(* Logix 5000 project; controller cal1615 1756-L62 rev 16.20; software revision 16.05; part 26 of 78 *)
(* tags used below, declared in another part *)
   AFI : BOOL;   // Always False Bit
   FAULT : BOOL;   // Fault AFI
   p01_param_fan_zero_speed : REAL;
   p01_param_open_oven_exh_sp : REAL;
   p01_recipe_active : recipe;   // Active Recipe
   p01r02 : routine;   // System Misc Control
   p01r09_open_oven : BOOL;
   p01r09_pb_global_reset : BOOL;   // System Modes PB: Global Fault Reset
   p02_dint_from_hmi : hmi_dint;
   p11r02_shutdown_temp : BOOL;   // Zone 1 Misc Control Safe Shutdown Temperature
   p11r30 : routine;   // Zone 1 Temperature Control
   p11r30_request_heat : BOOL;   // Zone 1 Temperature Control Request Heat
   p12_ai_exhaust_rpm : REAL;   // Zone 2 Analog Input Exhaust Fan RPM
   p12_ai_lfl : REAL;   // Zone 2 Analog Input Lower Flash Limit
   p12_ao_exhaust_selected_speed : REAL;   // Zone 2 Analog Output Exhaust Fan VFD Selected Speed
   p12_di_burner_auto : BOOL;   // Zone 2 Digital Input Burner Auto
   p12_di_exh : acs800_di_normal;   // Zone 2 Digital Inputs Exhaust Fan
   p12_di_exh_fan_mtr_ts : BOOL;   // Zone 2 Digital Input Exhaust Fan Motor Thermostat OK
   p12_di_exh_flow_ok : BOOL;   // Zone 2 Digital Input Exhaust Flow OK
   p12_di_flame_on : BOOL;   // Zone 2 Digital Input Burner is On
   p12_di_fresh_air_clean : BOOL;   // Zone 2 Digital Input Fresh Air Filter Dirty
   p12_di_sp0 : BOOL;
   p12_di_tc01_bo : BOOL;   // Zone 2 Digital Input Control Thermocouple 1 Failure
   p12_di_tc02_bo : BOOL;   // Zone 2 Digital Input Control Thermocouple 2 Failure
   p12_di_zone_air_clean : BOOL;   // Zone 2 Digital Input Zone 2 Filter Dirty
   p12_do_exh : acs800_do_normal;   // Zone 2 Digital Output Exhaust Fan
   p12_param_lfl_hl : REAL;   // Zone 2 Parameter High LFL Limit
   p12_param_tc01_dev : REAL;   // Zone 2 Parameter Oven Temperature Deviation from Setpoint
   p12r01 : routine;   // Zone 2 Main
   p12r02_shutdown_temp : BOOL;   // Zone 2 Misc Control Safe Shutdown Temperature
   p12r20_safeties_ok : BOOL;   // Zone 2 Temperature Control Burner Safeties OK this Lightoff
   p12r20_state : DINT;   // Zone 2 Temperature Control State
   p12r30 : routine;   // Zone 2 Temperature Control
   p12r30_pb_zone_on : BOOL;   // Zone 2 Temperature Control PB: Start Zone Heat Control
   p12r30_pid_temp_sp_error : REAL;   // Zone 2 Temperature Control Setpoint/Process Variable Error (ABS)
   p12r30_request_deviation_warning : BOOL;   // Zone 2 Temperature Control Request Setpoint Deviation Warning
   p12r30_request_heat : BOOL;   // Zone 2 Temperature Control Request Heat
   p12r30_request_heat_last : BOOL;   // Zone 2 Temperature Control Request Heat Last Scan
   p12r30_request_manual : BOOL;   // Zone 2 Temperature Control Request Manual Control
   p12r30_timer_fault : TIMER[16];   // Zone 2 Temperature Control Fault Delay
   p12r30_timer_warning : TIMER[12];   // Zone 2 Temperature Control Warning Delay
   p12r31 : routine;   // Zone 2 Exhaust VFD
   p12r31_pb_start : BOOL;   // Zone 2 Exhaust VFD PB: Start
   p12r31_pb_stop : BOOL;   // Zone 2 Exhaust VFD PB: Stop
   p12r31_request_auto_run : BOOL;   // Zone 2 Exhaust Fan Run Request
   p12r31_run_permissive : BOOL;   // Zone 2 Exhaust VFD Run Permissive
   p12r31_timer_fault : TIMER[5];   // Zone 2 Exhaust VFD Fault Timer
   p12r31_timer_warning : TIMER[5];   // Zone 2 Exhaust VFD Waringing Timer
   p12r31_vfd_stopped : BOOL;   // Zone 2 Exhaust VFD VFD Stopped
   p23_di_exhaust_speed_ok : BOOL;
   p23_di_supply_speed_ok : BOOL;
   p23r02 : routine;   // Impreg Misc Control
(* P12_Zone_2, continued *)

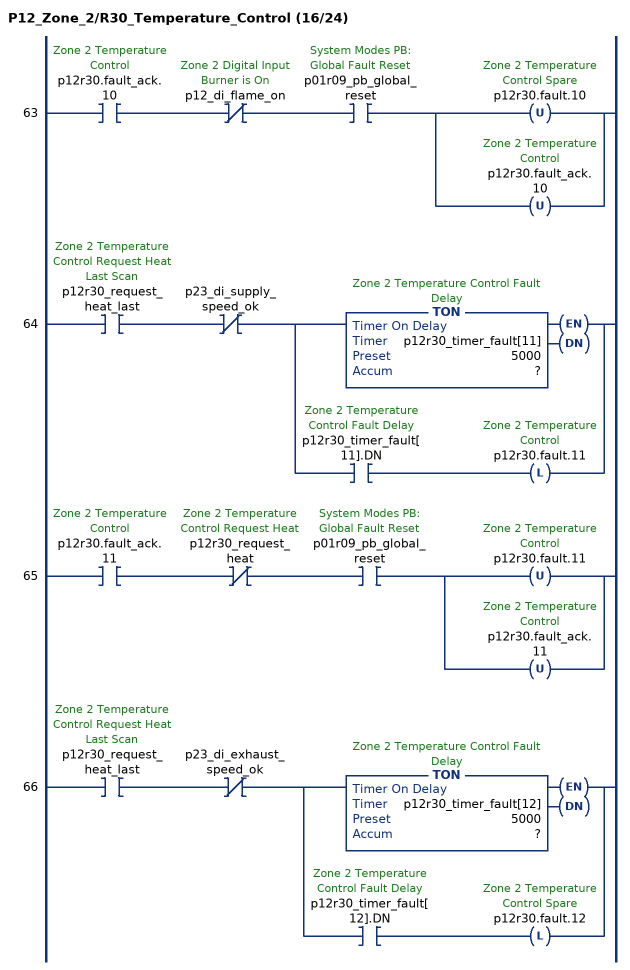
   [picture p454: P12_Zone_2/R30_Temperature_Control rungs 63-66]
   63: XIC(p12r30.fault_ack.10)XIO(p12_di_flame_on)XIC(p01r09_pb_global_reset)[OTU(p12r30.fault.10) ,OTU(p12r30.fault_ack.10) ];
   64: XIC(p12r30_request_heat_last)XIO(p23_di_supply_speed_ok)[TON(p12r30_timer_fault[11],?,?) ,XIC(p12r30_timer_fault[11].DN) OTL(p12r30.fault.11) ];
   65: XIC(p12r30.fault_ack.11)XIO(p12r30_request_heat)XIC(p01r09_pb_global_reset)[OTU(p12r30.fault.11) ,OTU(p12r30.fault_ack.11) ];
   66: XIC(p12r30_request_heat_last)XIO(p23_di_exhaust_speed_ok)[TON(p12r30_timer_fault[12],?,?) ,XIC(p12r30_timer_fault[12].DN) OTL(p12r30.fault.12) ];
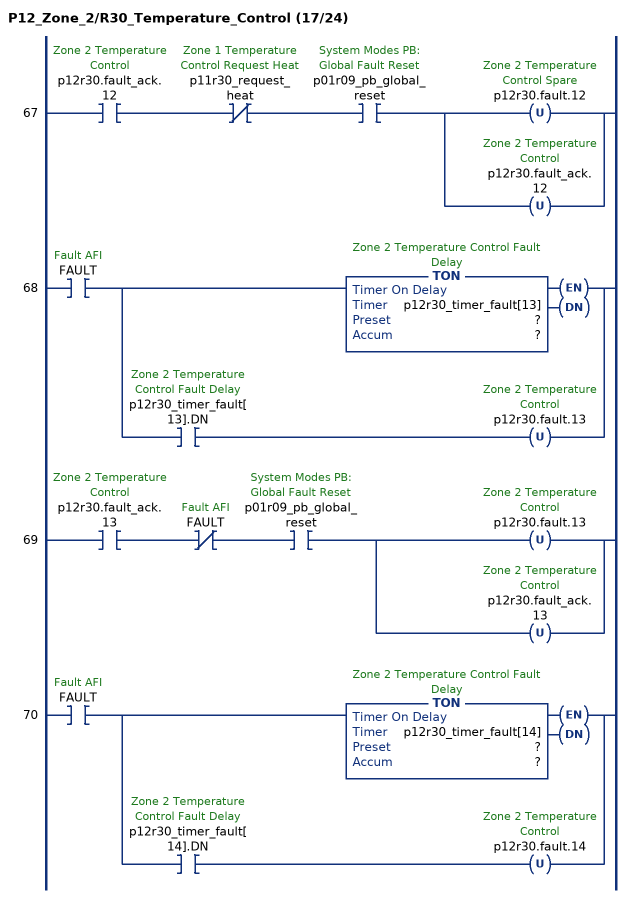
   67: XIC(p12r30.fault_ack.12)XIO(p11r30_request_heat)XIC(p01r09_pb_global_reset)[OTU(p12r30.fault.12) ,OTU(p12r30.fault_ack.12) ];
   68: XIC(FAULT)[TON(p12r30_timer_fault[13],?,?) ,XIC(p12r30_timer_fault[13].DN) OTU(p12r30.fault.13) ];
   69: XIC(p12r30.fault_ack.13)XIO(FAULT)XIC(p01r09_pb_global_reset)[OTU(p12r30.fault.13) ,OTU(p12r30.fault_ack.13) ];
   70: XIC(FAULT)[TON(p12r30_timer_fault[14],?,?) ,XIC(p12r30_timer_fault[14].DN) OTU(p12r30.fault.14) ];
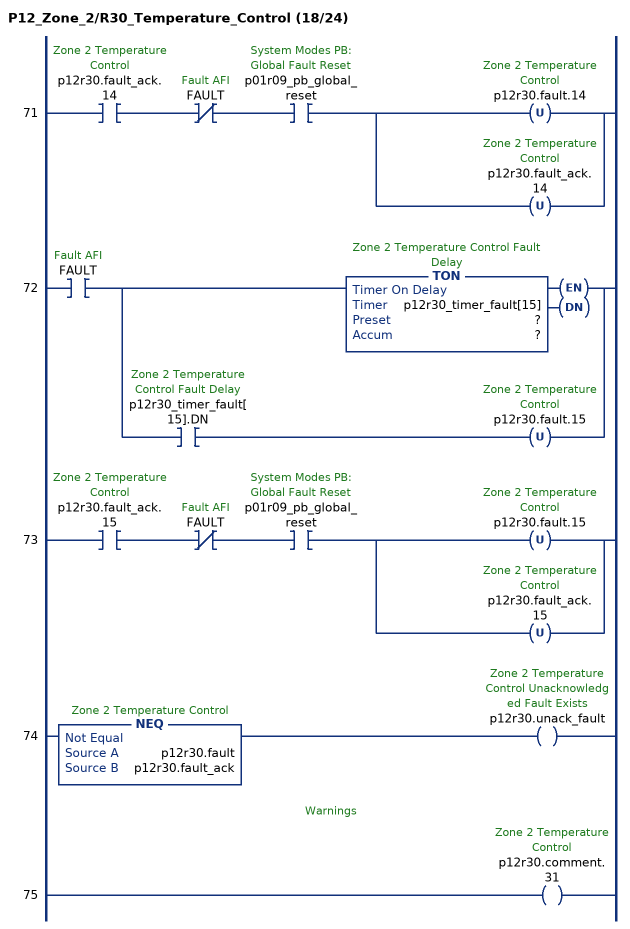
   71: XIC(p12r30.fault_ack.14)XIO(FAULT)XIC(p01r09_pb_global_reset)[OTU(p12r30.fault.14) ,OTU(p12r30.fault_ack.14) ];
   72: XIC(FAULT)[TON(p12r30_timer_fault[15],?,?) ,XIC(p12r30_timer_fault[15].DN) OTU(p12r30.fault.15) ];
   73: XIC(p12r30.fault_ack.15)XIO(FAULT)XIC(p01r09_pb_global_reset)[OTU(p12r30.fault.15) ,OTU(p12r30.fault_ack.15) ];
   74: NEQ(p12r30.fault,p12r30.fault_ack)OTE(p12r30.unack_fault);
   // Warnings
   75: OTE(p12r30.comment.31);
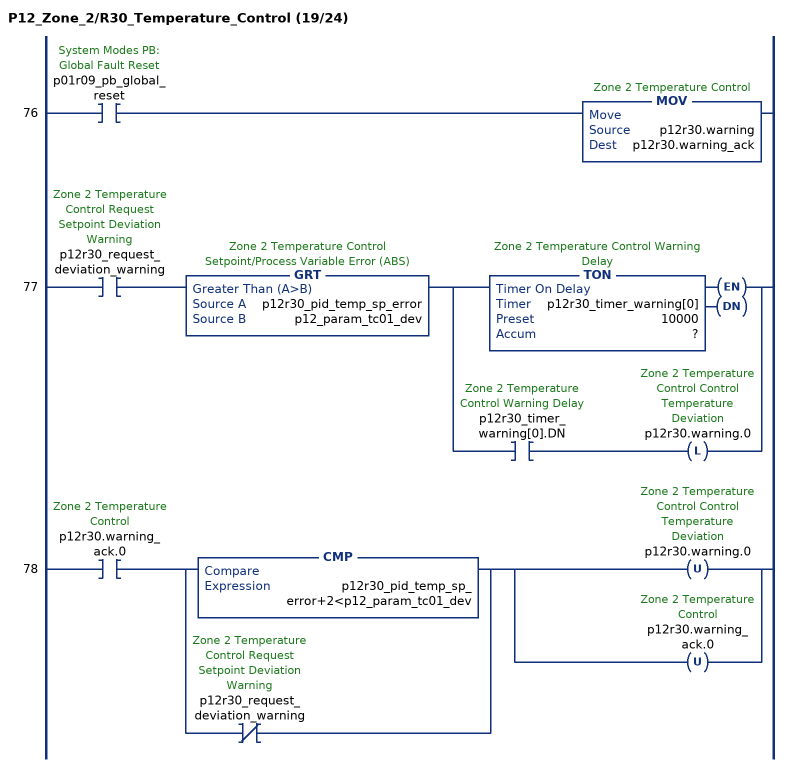
   76: XIC(p01r09_pb_global_reset)MOV(p12r30.warning,p12r30.warning_ack);
   77: XIC(p12r30_request_deviation_warning)GRT(p12r30_pid_temp_sp_error,p12_param_tc01_dev)[TON(p12r30_timer_warning[0],?,?) ,XIC(p12r30_timer_warning[0].DN) OTL(p12r30.warning.0) ];
   78: XIC(p12r30.warning_ack.0)[CMP(p12r30_pid_temp_sp_error+2<p12_param_tc01_dev) ,XIO(p12r30_request_deviation_warning) ][OTU(p12r30.warning.0) ,OTU(p12r30.warning_ack.0) ];
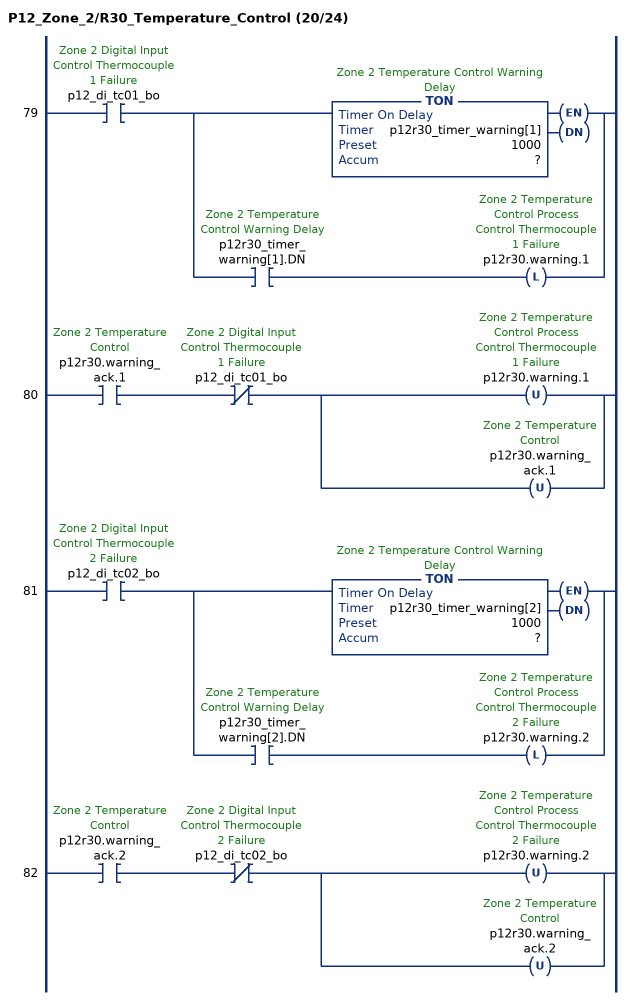
   79: XIC(p12_di_tc01_bo)[TON(p12r30_timer_warning[1],?,?) ,XIC(p12r30_timer_warning[1].DN) OTL(p12r30.warning.1) ];
   80: XIC(p12r30.warning_ack.1)XIO(p12_di_tc01_bo)[OTU(p12r30.warning.1) ,OTU(p12r30.warning_ack.1) ];
   81: XIC(p12_di_tc02_bo)[TON(p12r30_timer_warning[2],?,?) ,XIC(p12r30_timer_warning[2].DN) OTL(p12r30.warning.2) ];
   82: XIC(p12r30.warning_ack.2)XIO(p12_di_tc02_bo)[OTU(p12r30.warning.2) ,OTU(p12r30.warning_ack.2) ];
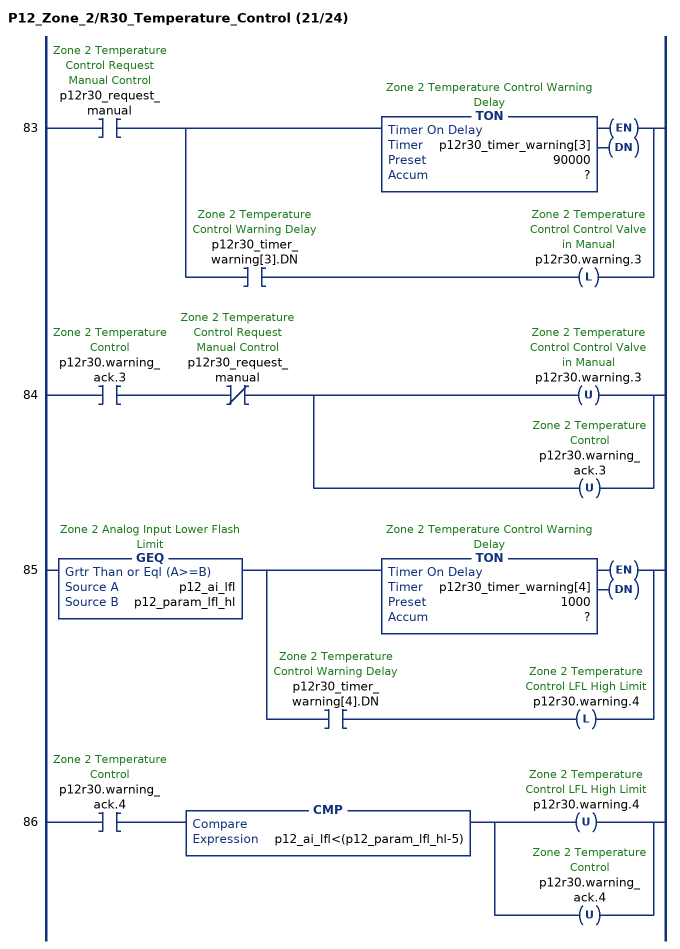
   83: XIC(p12r30_request_manual)[TON(p12r30_timer_warning[3],?,?) ,XIC(p12r30_timer_warning[3].DN) OTL(p12r30.warning.3) ];
   84: XIC(p12r30.warning_ack.3)XIO(p12r30_request_manual)[OTU(p12r30.warning.3) ,OTU(p12r30.warning_ack.3) ];
   85: GEQ(p12_ai_lfl,p12_param_lfl_hl)[TON(p12r30_timer_warning[4],?,?) ,XIC(p12r30_timer_warning[4].DN) OTL(p12r30.warning.4) ];
   86: XIC(p12r30.warning_ack.4)CMP(p12_ai_lfl<(p12_param_lfl_hl-5))[OTU(p12r30.warning.4) ,OTU(p12r30.warning_ack.4) ];
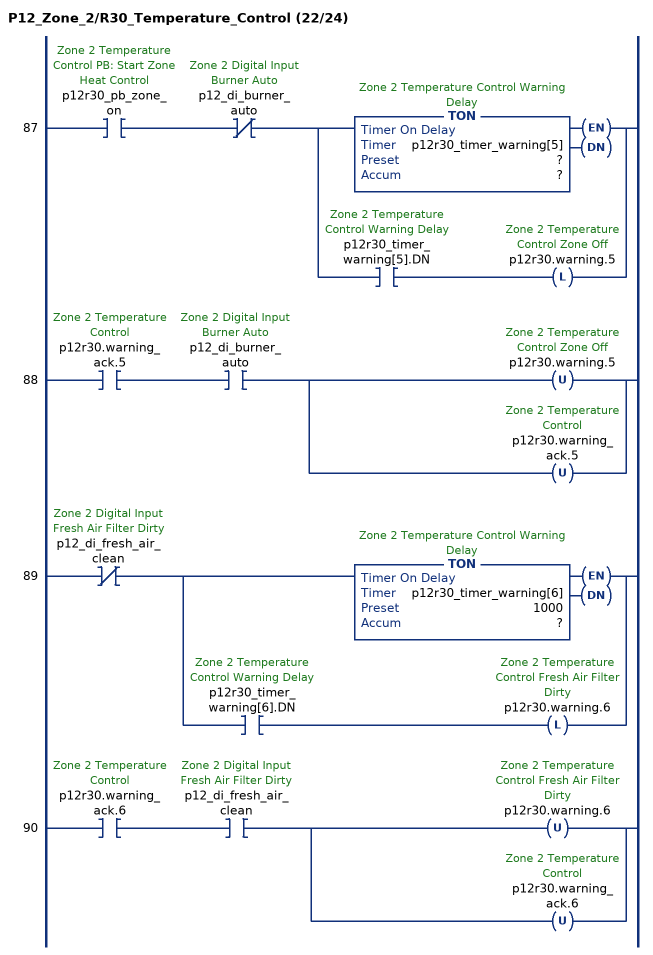
   87: XIC(p12r30_pb_zone_on)XIO(p12_di_burner_auto)[TON(p12r30_timer_warning[5],?,?) ,XIC(p12r30_timer_warning[5].DN) OTL(p12r30.warning.5) ];
   88: XIC(p12r30.warning_ack.5)XIC(p12_di_burner_auto)[OTU(p12r30.warning.5) ,OTU(p12r30.warning_ack.5) ];
   89: XIO(p12_di_fresh_air_clean)[TON(p12r30_timer_warning[6],?,?) ,XIC(p12r30_timer_warning[6].DN) OTL(p12r30.warning.6) ];
   90: XIC(p12r30.warning_ack.6)XIC(p12_di_fresh_air_clean)[OTU(p12r30.warning.6) ,OTU(p12r30.warning_ack.6) ];
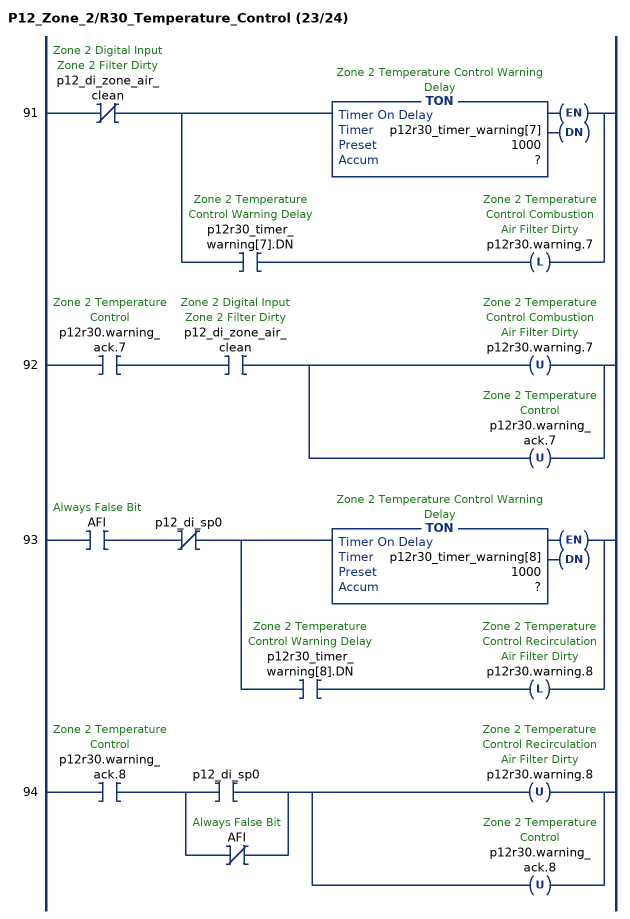
   91: XIO(p12_di_zone_air_clean)[TON(p12r30_timer_warning[7],?,?) ,XIC(p12r30_timer_warning[7].DN) OTL(p12r30.warning.7) ];
   92: XIC(p12r30.warning_ack.7)XIC(p12_di_zone_air_clean)[OTU(p12r30.warning.7) ,OTU(p12r30.warning_ack.7) ];
   93: XIC(AFI)XIO(p12_di_sp0)[TON(p12r30_timer_warning[8],?,?) ,XIC(p12r30_timer_warning[8].DN) OTL(p12r30.warning.8) ];
   94: XIC(p12r30.warning_ack.8)[XIC(p12_di_sp0) ,XIO(AFI) ][OTU(p12r30.warning.8) ,OTU(p12r30.warning_ack.8) ];
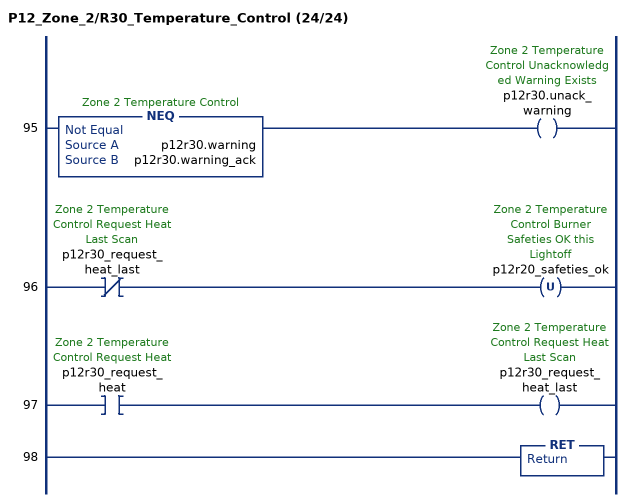
   95: NEQ(p12r30.warning,p12r30.warning_ack)OTE(p12r30.unack_warning);
   96: XIO(p12r30_request_heat_last)OTU(p12r20_safeties_ok);
   97: XIC(p12r30_request_heat)OTE(p12r30_request_heat_last);
   98: RET();
END_ROUTINE

ROUTINE R31_Exhaust_VFD   (* ladder *)
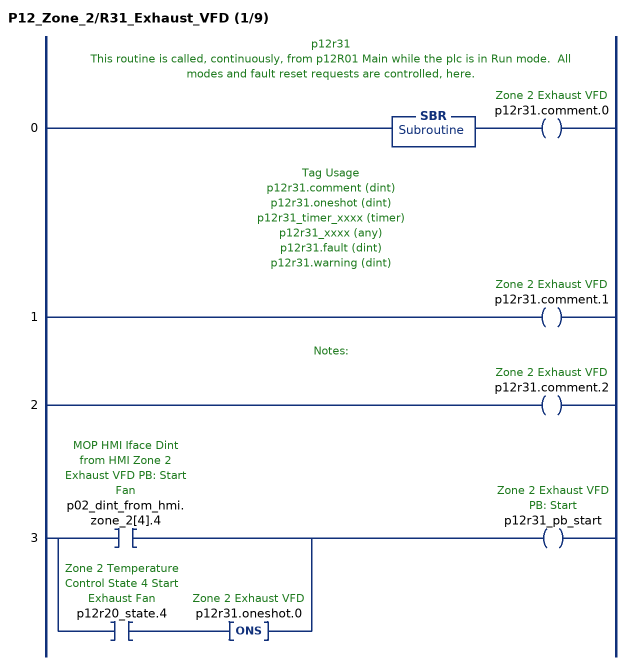
   // p12r31
   // This routine is called, continuously, from p12R01 Main while the plc is in Run mode.  All modes and fault reset requests are controlled, here.
   0: SBR()OTE(p12r31.comment.0);
   // Tag Usage
   // p12r31.comment (dint)
   // p12r31.oneshot (dint)
   // p12r31_timer_xxxx (timer)
   // p12r31_xxxx (any)
   // p12r31.fault (dint)
   // p12r31.warning (dint)
   1: OTE(p12r31.comment.1);
   // Notes:
   2: OTE(p12r31.comment.2);
   3: [XIC(p02_dint_from_hmi.zone_2[4].4) ,XIC(p12r20_state.4) ONS(p12r31.oneshot.0) ]OTE(p12r31_pb_start);
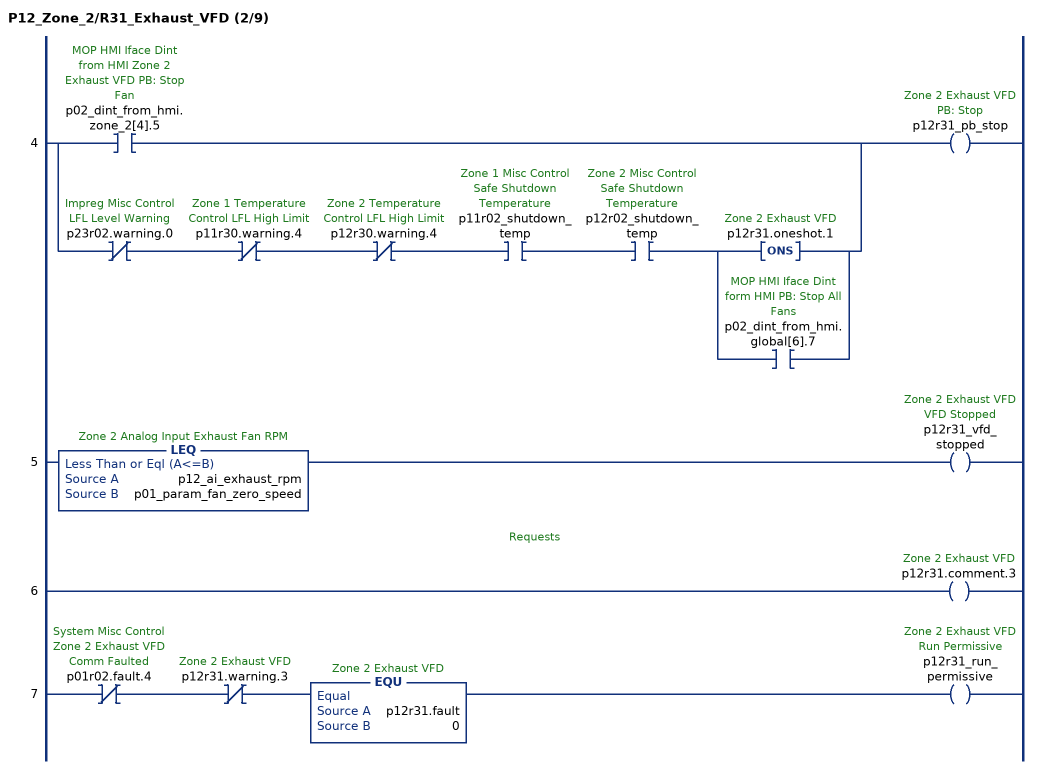
   4: [XIC(p02_dint_from_hmi.zone_2[4].5) ,XIO(p23r02.warning.0) XIO(p11r30.warning.4) XIO(p12r30.warning.4) XIC(p11r02_shutdown_temp) XIC(p12r02_shutdown_temp) [ONS(p12r31.oneshot.1) ,XIC(p02_dint_from_hmi.global[6].7) ] ]OTE(p12r31_pb_stop);
   5: LEQ(p12_ai_exhaust_rpm,p01_param_fan_zero_speed)OTE(p12r31_vfd_stopped);
   // Requests
   6: OTE(p12r31.comment.3);
   7: XIO(p01r02.fault.4)XIO(p12r31.warning.3)EQU(p12r31.fault,0)OTE(p12r31_run_permissive);
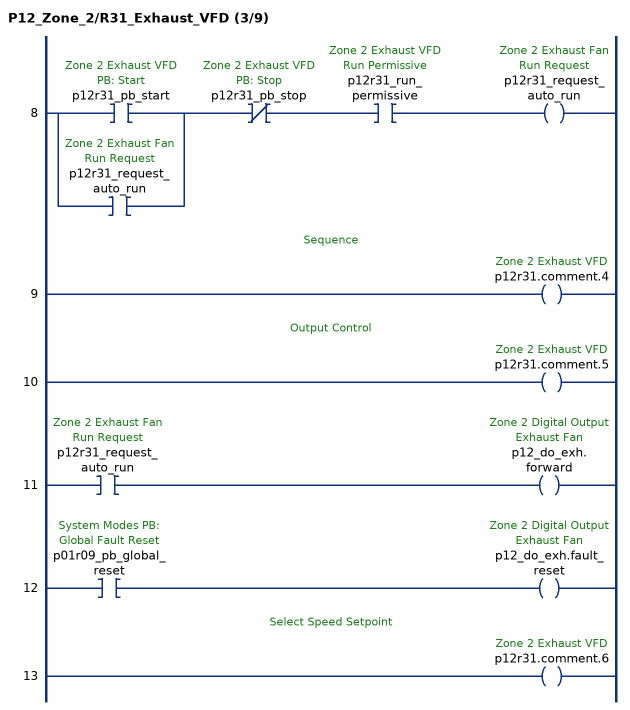
   8: [XIC(p12r31_pb_start) ,XIC(p12r31_request_auto_run) ]XIO(p12r31_pb_stop)XIC(p12r31_run_permissive)OTE(p12r31_request_auto_run);
   // Sequence
   9: OTE(p12r31.comment.4);
   // Output Control
   10: OTE(p12r31.comment.5);
   11: XIC(p12r31_request_auto_run)OTE(p12_do_exh.forward);
   12: XIC(p01r09_pb_global_reset)OTE(p12_do_exh.fault_reset);
   // Select Speed Setpoint
   13: OTE(p12r31.comment.6);
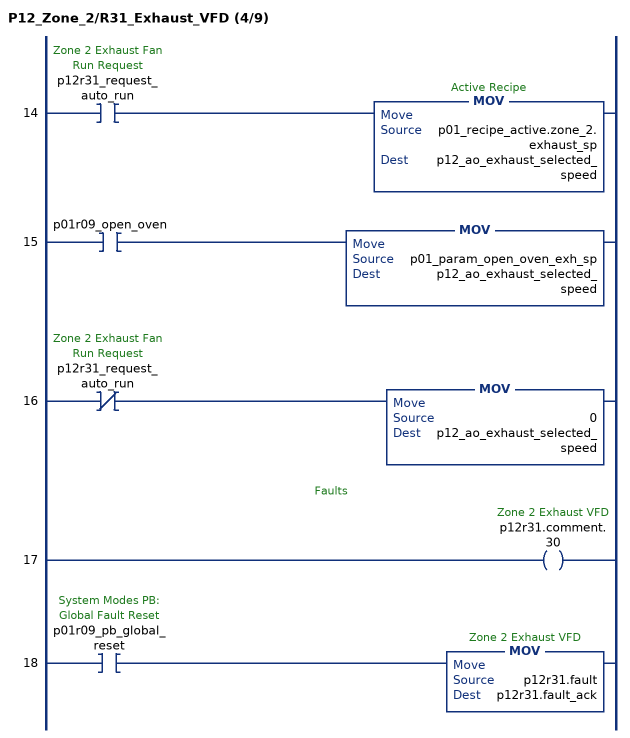
   14: XIC(p12r31_request_auto_run)MOV(p01_recipe_active.zone_2.exhaust_sp,p12_ao_exhaust_selected_speed);
   15: XIC(p01r09_open_oven)MOV(p01_param_open_oven_exh_sp,p12_ao_exhaust_selected_speed);
   16: XIO(p12r31_request_auto_run)MOV(0,p12_ao_exhaust_selected_speed);
   // Faults
   17: OTE(p12r31.comment.30);
   18: XIC(p01r09_pb_global_reset)MOV(p12r31.fault,p12r31.fault_ack);
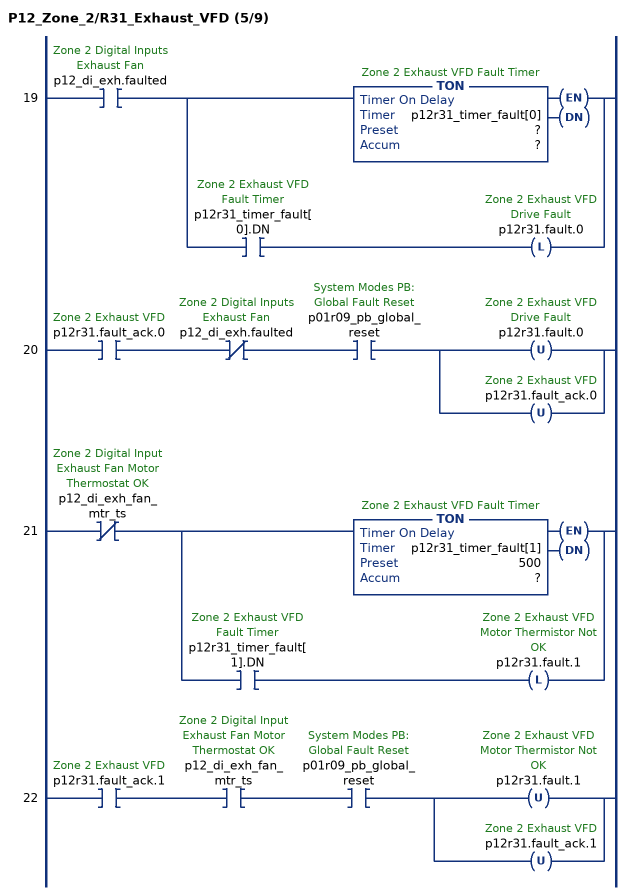
   19: XIC(p12_di_exh.faulted)[TON(p12r31_timer_fault[0],?,?) ,XIC(p12r31_timer_fault[0].DN) OTL(p12r31.fault.0) ];
   20: XIC(p12r31.fault_ack.0)XIO(p12_di_exh.faulted)XIC(p01r09_pb_global_reset)[OTU(p12r31.fault.0) ,OTU(p12r31.fault_ack.0) ];
   21: XIO(p12_di_exh_fan_mtr_ts)[TON(p12r31_timer_fault[1],?,?) ,XIC(p12r31_timer_fault[1].DN) OTL(p12r31.fault.1) ];
   22: XIC(p12r31.fault_ack.1)XIC(p12_di_exh_fan_mtr_ts)XIC(p01r09_pb_global_reset)[OTU(p12r31.fault.1) ,OTU(p12r31.fault_ack.1) ];
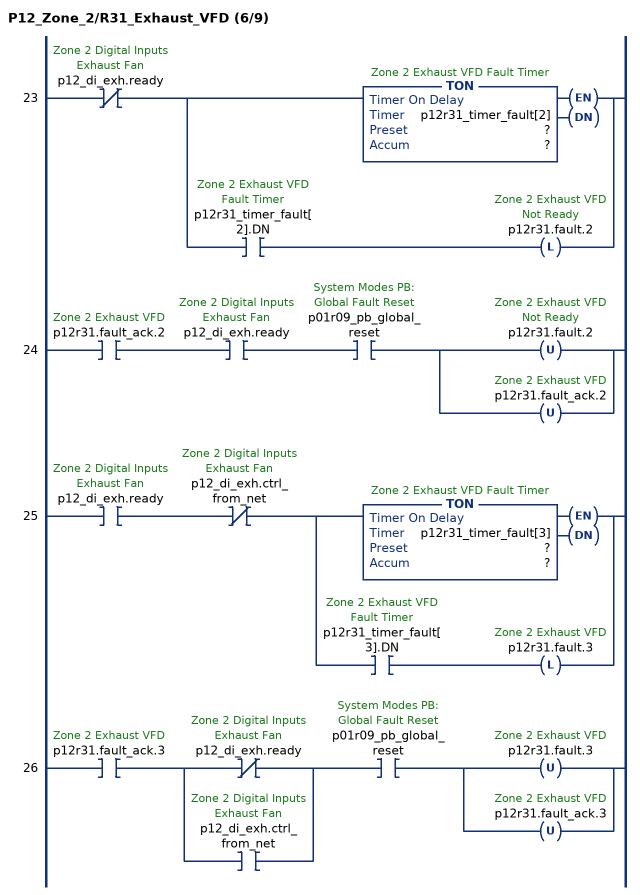
   23: XIO(p12_di_exh.ready)[TON(p12r31_timer_fault[2],?,?) ,XIC(p12r31_timer_fault[2].DN) OTL(p12r31.fault.2) ];
   24: XIC(p12r31.fault_ack.2)XIC(p12_di_exh.ready)XIC(p01r09_pb_global_reset)[OTU(p12r31.fault.2) ,OTU(p12r31.fault_ack.2) ];
   25: XIC(p12_di_exh.ready)XIO(p12_di_exh.ctrl_from_net)[TON(p12r31_timer_fault[3],?,?) ,XIC(p12r31_timer_fault[3].DN) OTL(p12r31.fault.3) ];
   26: XIC(p12r31.fault_ack.3)[XIO(p12_di_exh.ready) ,XIC(p12_di_exh.ctrl_from_net) ]XIC(p01r09_pb_global_reset)[OTU(p12r31.fault.3) ,OTU(p12r31.fault_ack.3) ];
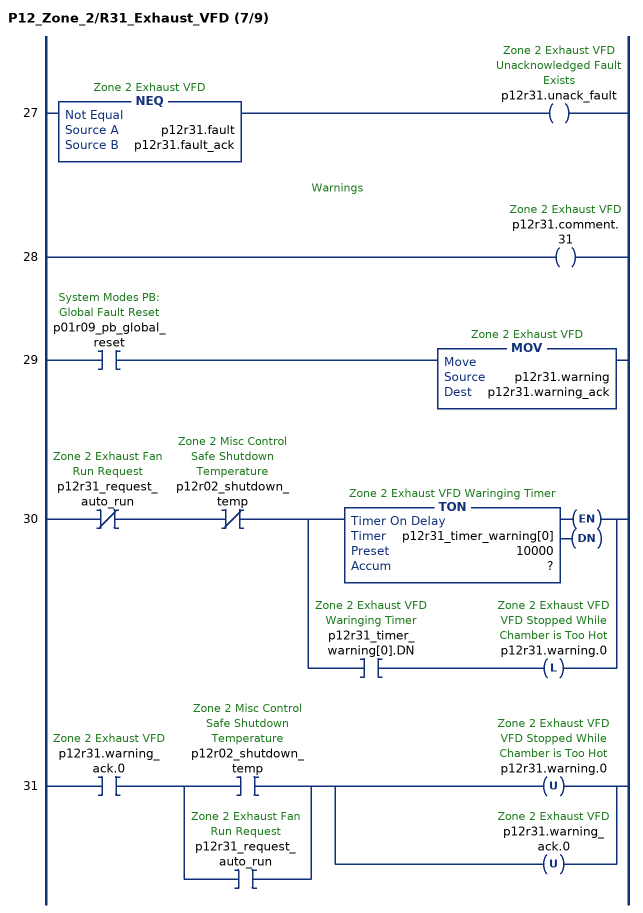
   27: NEQ(p12r31.fault,p12r31.fault_ack)OTE(p12r31.unack_fault);
   // Warnings
   28: OTE(p12r31.comment.31);
   29: XIC(p01r09_pb_global_reset)MOV(p12r31.warning,p12r31.warning_ack);
   30: XIO(p12r31_request_auto_run)XIO(p12r02_shutdown_temp)[TON(p12r31_timer_warning[0],?,?) ,XIC(p12r31_timer_warning[0].DN) OTL(p12r31.warning.0) ];
   31: XIC(p12r31.warning_ack.0)[XIC(p12r02_shutdown_temp) ,XIC(p12r31_request_auto_run) ][OTU(p12r31.warning.0) ,OTU(p12r31.warning_ack.0) ];
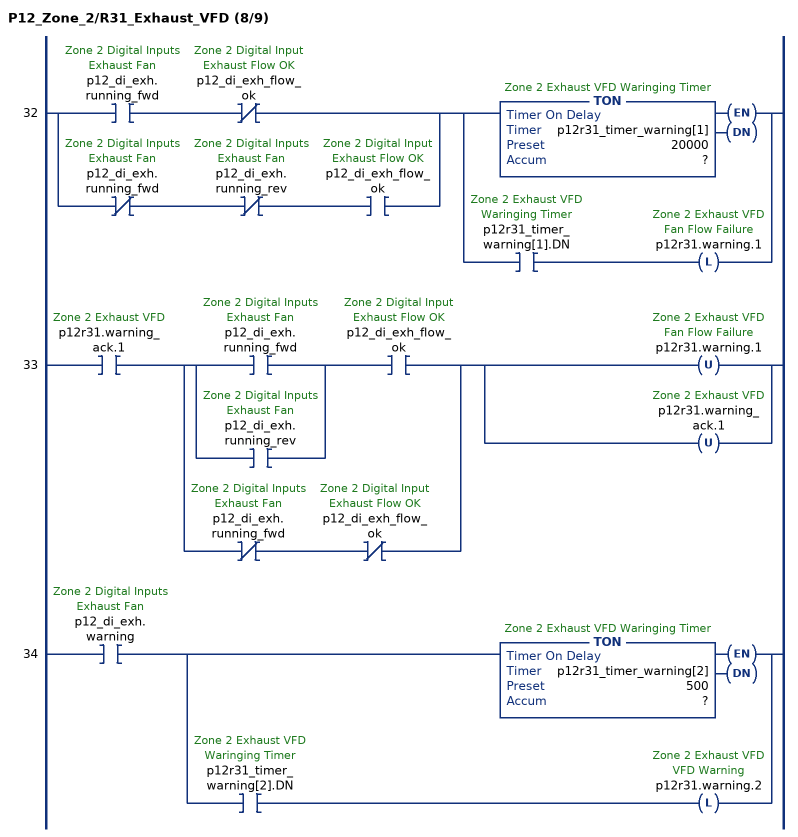
   32: [XIC(p12_di_exh.running_fwd) XIO(p12_di_exh_flow_ok) ,XIO(p12_di_exh.running_fwd) XIO(p12_di_exh.running_rev) XIC(p12_di_exh_flow_ok) ][TON(p12r31_timer_warning[1],?,?) ,XIC(p12r31_timer_warning[1].DN) OTL(p12r31.warning.1) ];
   33: XIC(p12r31.warning_ack.1)[[XIC(p12_di_exh.running_fwd) ,XIC(p12_di_exh.running_rev) ] XIC(p12_di_exh_flow_ok) ,XIO(p12_di_exh.running_fwd) XIO(p12_di_exh_flow_ok) ][OTU(p12r31.warning.1) ,OTU(p12r31.warning_ack.1) ];
   34: XIC(p12_di_exh.warning)[TON(p12r31_timer_warning[2],?,?) ,XIC(p12r31_timer_warning[2].DN) OTL(p12r31.warning.2) ];
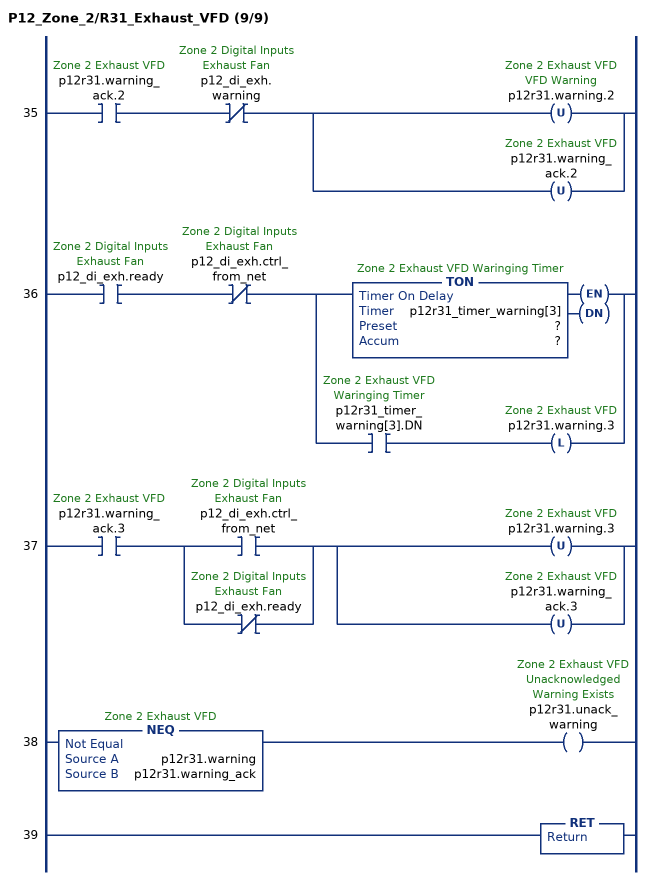
   35: XIC(p12r31.warning_ack.2)XIO(p12_di_exh.warning)[OTU(p12r31.warning.2) ,OTU(p12r31.warning_ack.2) ];
   36: XIC(p12_di_exh.ready)XIO(p12_di_exh.ctrl_from_net)[TON(p12r31_timer_warning[3],?,?) ,XIC(p12r31_timer_warning[3].DN) OTL(p12r31.warning.3) ];
   37: XIC(p12r31.warning_ack.3)[XIC(p12_di_exh.ctrl_from_net) ,XIO(p12_di_exh.ready) ][OTU(p12r31.warning.3) ,OTU(p12r31.warning_ack.3) ];
   38: NEQ(p12r31.warning,p12r31.warning_ack)OTE(p12r31.unack_warning);
   39: RET();
END_ROUTINE
